// TIA Portal V16 export
// export: Created 2022-11-14T17:35:47.2459198Z, ExportSetting WithDefaults, DisplayName Totally Integrated Automation Portal, DisplayVersion V16, DisplayName TIA Portal Version Control Interface, DisplayVersion V16, DisplayName TIA Portal Openness, DisplayVersion V16, DisplayName STEP 7 Professional, DisplayVersion V16, DisplayName STEP 7 Safety, DisplayVersion V16, DisplayName WinCC Advanced, DisplayVersion V16
DATA_BLOCK "DB238_Program12"   // DB238
{ S7_Optimized_Access := 'FALSE' }
AUTHOR : Robopac
VERSION : 0.0
// stored: AutoNumber false, IsOnlyStoredInLoadMemory false, IsWriteProtectedInAS false
   VAR RETAIN
      Program12 { S7_SetPoint := 'True'} : "DatiProgramma";
   END_VAR
BEGIN
   Program12.Wrapping := TRUE;
   Program12.TopLenght := 500;
   Program12.TopRelease := 0;
   Program12.TopDown := 0;
   Program12.Top := 4;
   Program12.PressurePTime := 0;
   Program12.LifterTime := 0;
   Program12.RevOverContrast := 1;
   Program12.RopeEndCycle := 16#02;
   Program12.Spare4 := 16#01;
   Program12.RopeTime := 1500;
   Program12.RevOverClamp := 1;
   Program12.FilmForceFinalRev := 10;
   Program12.FilmPrestretchFinalRev := 100;
   Program12.ArmSpeed := 100;
   Program12.CarriageDown4Top := 500;
   Program12.TopDownTime := 1500;
   Program12.LapsUnderTop := 0;
   Program12.Spare6 := 0;
   Program12.Spare7 := 0;
   Program12.Spare8 := 0;
   Program12.Spare9 := 0;
   Program12.Spare10 := 0;
   Program12.Spare11 := 0;
   Program12.Spare12 := 0;
   Program12.Overlap0_1 := 0;
   Program12.Height1 := 130;
   Program12.Landmark1 := FALSE;
   Program12.Lifter1 := FALSE;
   Program12.SpareBit1H1 := FALSE;
   Program12.Airblower1 := TRUE;
   Program12.NextStep1 := TRUE;
   Program12.PressureP1 := TRUE;
   Program12.SpareByte2H1 := 16#00;
   Program12.Revolution1 := 1;
   Program12.RopeUnit1_1 := 16#01;
   Program12.RopeUnit1_2 := 16#01;
   Program12.FilmForce1 := 5;
   Program12.FilmPrestretch1 := 200;
   Program12.Spare3H1 := 0;
   Program12.Spare49 := 0;
   Program12.Spare50 := 0;
   Program12.Spare51 := 0;
   Program12.Spare52 := 0;
   Program12.Spare53 := 0;
   Program12.Overlap1_2 := 0;
   Program12.Height2 := 50;
   Program12.Landmark2 := FALSE;
   Program12.Lifter2 := FALSE;
   Program12.SpareBit1H2 := FALSE;
   Program12.Airblower2 := TRUE;
   Program12.NextStep2 := TRUE;
   Program12.PressureP2 := TRUE;
   Program12.SpareByte2H2 := 16#00;
   Program12.Revolution2 := 1;
   Program12.RopeUnit2_1 := 16#01;
   Program12.RopeUnit2_2 := 16#01;
   Program12.FilmForce2 := 20;
   Program12.FilmPrestretch2 := 200;
   Program12.Spare3H2 := 0;
   Program12.Spare54 := 0;
   Program12.Spare55 := 0;
   Program12.Spare56 := 0;
   Program12.Spare57 := 0;
   Program12.Spare58 := 0;
   Program12.Overlap2_3 := 100;
   Program12.Height3 := -50;
   Program12.Landmark3 := TRUE;
   Program12.Lifter3 := FALSE;
   Program12.SpareBit1H3 := FALSE;
   Program12.Airblower3 := TRUE;
   Program12.NextStep3 := TRUE;
   Program12.PressureP3 := TRUE;
   Program12.SpareByte2H3 := 16#00;
   Program12.Revolution3 := 2;
   Program12.RopeUnit3_1 := 16#01;
   Program12.RopeUnit3_2 := 16#01;
   Program12.FilmForce3 := 30;
   Program12.FilmPrestretch3 := 200;
   Program12.Spare3H3 := 0;
   Program12.Spare59 := 0;
   Program12.Spare60 := 0;
   Program12.Spare61 := 380;
   Program12.Spare62 := 2800;
   Program12.Spare63 := 0;
   Program12.Overlap3_4 := 100;
   Program12.Height4 := 100;
   Program12.Landmark4 := FALSE;
   Program12.Lifter4 := FALSE;
   Program12.SpareBit1H4 := FALSE;
   Program12.Airblower4 := TRUE;
   Program12.NextStep4 := TRUE;
   Program12.PressureP4 := TRUE;
   Program12.SpareByte2H4 := 16#00;
   Program12.Revolution4 := 3;
   Program12.RopeUnit4_1 := 16#02;
   Program12.RopeUnit4_2 := 16#02;
   Program12.FilmForce4 := 30;
   Program12.FilmPrestretch4 := 200;
   Program12.Spare3H4 := 0;
   Program12.Spare64 := 0;
   Program12.Spare65 := 0;
   Program12.Spare66 := 0;
   Program12.Spare67 := 0;
   Program12.Spare68 := 0;
   Program12.Overlap4_5 := 0;
   Program12.Height5 := 50;
   Program12.Landmark5 := FALSE;
   Program12.Lifter5 := FALSE;
   Program12.SpareBit1H5 := FALSE;
   Program12.Airblower5 := TRUE;
   Program12.NextStep5 := FALSE;
   Program12.PressureP5 := FALSE;
   Program12.SpareByte2H5 := 16#00;
   Program12.Revolution5 := 1;
   Program12.RopeUnit5_1 := 16#01;
   Program12.RopeUnit5_2 := 16#01;
   Program12.FilmForce5 := 30;
   Program12.FilmPrestretch5 := 200;
   Program12.Spare3H5 := 0;
   Program12.Spare69 := 0;
   Program12.Spare70 := 0;
   Program12.Spare71 := 0;
   Program12.Spare72 := 0;
   Program12.Spare73 := 0;
   Program12.Overlap5_6 := 100;
   Program12.Height6 := 50;
   Program12.Landmark6 := FALSE;
   Program12.Lifter6 := FALSE;
   Program12.SpareBit1H6 := FALSE;
   Program12.Airblower6 := TRUE;
   Program12.NextStep6 := FALSE;
   Program12.PressureP6 := FALSE;
   Program12.SpareByte2H6 := 16#00;
   Program12.Revolution6 := 2;
   Program12.RopeUnit6_1 := 16#02;
   Program12.RopeUnit6_2 := 16#01;
   Program12.FilmForce6 := 20;
   Program12.FilmPrestretch6 := 200;
   Program12.Spare3H6 := 0;
   Program12.Spare74 := 0;
   Program12.Spare75 := 0;
   Program12.Spare76 := 0;
   Program12.Spare77 := 0;
   Program12.Spare78 := 0;
   Program12.Overlap6_7 := 0;
   Program12.Height7 := 0;
   Program12.Landmark7 := FALSE;
   Program12.Lifter7 := FALSE;
   Program12.SpareBit1H7 := FALSE;
   Program12.Airblower7 := FALSE;
   Program12.NextStep7 := TRUE;
   Program12.PressureP7 := FALSE;
   Program12.SpareByte2H7 := 16#00;
   Program12.Revolution7 := 1;
   Program12.RopeUnit7_1 := 16#01;
   Program12.RopeUnit7_2 := 16#01;
   Program12.FilmForce7 := 0;
   Program12.FilmPrestretch7 := 100;
   Program12.Spare3H7 := 0;
   Program12.Spare79 := 0;
   Program12.Spare80 := 0;
   Program12.Spare81 := 0;
   Program12.Spare82 := 0;
   Program12.Spare83 := 0;
   Program12.Overlap7_8 := 0;
   Program12.Height8 := 0;
   Program12.Landmark8 := FALSE;
   Program12.Lifter8 := FALSE;
   Program12.SpareBit1H8 := FALSE;
   Program12.Airblower8 := FALSE;
   Program12.NextStep8 := TRUE;
   Program12.PressureP8 := FALSE;
   Program12.SpareByte2H8 := 16#00;
   Program12.Revolution8 := 1;
   Program12.RopeUnit8_1 := 16#01;
   Program12.RopeUnit8_2 := 16#01;
   Program12.FilmForce8 := 0;
   Program12.FilmPrestretch8 := 100;
   Program12.Spare3H8 := 0;
   Program12.Spare84 := 0;
   Program12.Spare85 := 0;
   Program12.Spare86 := 0;
   Program12.Spare87 := 0;
   Program12.Spare88 := 0;
   Program12.Overlap8_9 := 0;
   Program12.Height9 := 0;
   Program12.Landmark9 := FALSE;
   Program12.Lifter9 := FALSE;
   Program12.SpareBit1H9 := FALSE;
   Program12.Airblower9 := FALSE;
   Program12.NextStep9 := TRUE;
   Program12.PressureP9 := FALSE;
   Program12.SpareByte2H9 := 16#00;
   Program12.Revolution9 := 1;
   Program12.RopeUnit9_1 := 16#01;
   Program12.RopeUnit9_2 := 16#01;
   Program12.FilmForce9 := 0;
   Program12.FilmPrestretch9 := 100;
   Program12.Spare3H9 := 0;
   Program12.Spare89 := 0;
   Program12.Spare90 := 0;
   Program12.Spare91 := 0;
   Program12.Spare92 := 0;
   Program12.Spare93 := 0;
   Program12.Overlap9_10 := 0;
   Program12.Height10 := 0;
   Program12.Landmark10 := FALSE;
   Program12.Lifter10 := FALSE;
   Program12.SpareBit1H10 := FALSE;
   Program12.Airblower10 := FALSE;
   Program12.NextStep10 := FALSE;
   Program12.PressureP10 := FALSE;
   Program12.SpareByte2H10 := 16#00;
   Program12.Revolution10 := 1;
   Program12.RopeUnit10_1 := 16#01;
   Program12.RopeUnit10_2 := 16#01;
   Program12.FilmForce10 := 0;
   Program12.FilmPrestretch10 := 100;
   Program12.Spare3H10 := 0;
   Program12.Spare94 := 0;
   Program12.Spare95 := 0;
   Program12.Spare96 := 0;
   Program12.Spare97 := 0;
   Program12.Spare98 := 0;
   Program12.Overlap10_11 := 0;
   Program12.Height11 := 0;
   Program12.Landmark11 := FALSE;
   Program12.Lifter11 := FALSE;
   Program12.SpareBit1H11 := FALSE;
   Program12.Airblower11 := FALSE;
   Program12.NextStep11 := TRUE;
   Program12.PressureP11 := FALSE;
   Program12.SpareByte2H11 := 16#00;
   Program12.Revolution11 := 1;
   Program12.RopeUnit11_1 := 16#01;
   Program12.RopeUnit11_2 := 16#01;
   Program12.FilmForce11 := 0;
   Program12.FilmPrestretch11 := 100;
   Program12.Spare3H11 := 0;
   Program12.Spare99 := 0;
   Program12.Spare100 := 0;
   Program12.Spare101 := 0;
   Program12.Spare102 := 0;
   Program12.Spare103 := 0;
   Program12.Overlap11_12 := 0;
   Program12.Height12 := 0;
   Program12.Landmark12 := FALSE;
   Program12.Lifter12 := FALSE;
   Program12.SpareBit1H12 := FALSE;
   Program12.Airblower12 := FALSE;
   Program12.NextStep12 := FALSE;
   Program12.PressureP12 := FALSE;
   Program12.SpareByte2H12 := 16#00;
   Program12.Revolution12 := 1;
   Program12.RopeUnit12_1 := 16#01;
   Program12.RopeUnit12_2 := 16#01;
   Program12.FilmForce12 := 0;
   Program12.FilmPrestretch12 := 100;
   Program12.Spare3H12 := 0;
   Program12.Spare104 := 0;
   Program12.Spare105 := 0;
   Program12.Spare106 := 0;
   Program12.Spare107 := 0;
   Program12.Spare108 := 0;
END_DATA_BLOCK
